{attribute 'qualified_only'}
{attribute 'strict'}
TYPE InternalState :
(
	passive := 0,
	override := 1,
	udpOnly := 2
);
END_TYPE

(* stored: Version 1.1.0.1, ProductVersion 3.1.4022.18
   DUT InternalState: Id {884ec536-736f-4bab-833f-b6970f84051f} *)
